{attribute 'GeneratedUsingTerminal: EL3446-0000-0016'}
{attribute addProperty BoxType "EL3446-0000-0016"}
{attribute addProperty Id "I1_CurrentAT %I*I1_Current_AFE1DFA29I2_CurrentAT %I*I2_Current_AFE1DFA29I3_CurrentAT %I*I3_Current_AFE1DFA29I4_CurrentAT %I*I4_Current_AFE1DFA29I5_CurrentAT %I*I5_Current_AFE1DFA29I6_CurrentAT %I*I6_Current_AFE1DFA29WcStateAT %I*WcState_9091E0EB2InfoDataAT %I*InfoData_BEF6B88E18"}
{attribute addProperty CRC "3645717692"}
{attribute addProperty Size "74"}
TYPE EL3446_D94D3CBC EXTENDS EtcSlaveTerminalBase_947E5A46 :
STRUCT
	{attribute addProperty Name "I1_Current"}
	I1_Current : I1_Current_AFE1DFA2;
	{attribute addProperty Name "I2_Current"}
	I2_Current : I2_Current_AFE1DFA2;
	{attribute addProperty Name "I3_Current"}
	I3_Current : I3_Current_AFE1DFA2;
	{attribute addProperty Name "I4_Current"}
	I4_Current : I4_Current_AFE1DFA2;
	{attribute addProperty Name "I5_Current"}
	I5_Current : I5_Current_AFE1DFA2;
	{attribute addProperty Name "I6_Current"}
	I6_Current : I6_Current_AFE1DFA2;
	{attribute addProperty Name "WcState"}
	WcState : WcState_9091E0EB;
	{attribute addProperty Name "InfoData"}
	InfoData : InfoData_BEF6B88E;
END_STRUCT
END_TYPE

(* stored: Version 1.2.0.0, ProductVersion 3.1.4024.9
   DUT EL3446_D94D3CBC: Id {512bbec3-cd86-46bb-ac30-6008b786cd0a} *)
